FUNCTION_BLOCK FB_HVPS EXTENDS FB_HMIBase
VAR
	hvps : REFERENCE TO FB_HVPS_System;  // Reference to avoid copying and allow validation
	hvpsStatus : ARRAY[GC_HVPS.INDEX_SUPPLY_MIN..GC_HVPS.INDEX_SUPPLY_MAX] OF ST_HMIHvpsStatus;  // Status for all 4 supplies
END_VAR

METHOD ClearErrors : BOOL
VAR_INPUT
	index : DINT;
END_VAR
// Clear errors for specified supply
IF __ISVALIDREF(hvps) THEN
	hvps.ClearErrors(index);
	ClearErrors := TRUE;
END_IF
END_METHOD

METHOD Cyclic
VAR
	i : DINT;
	status : ARRAY[GC_HVPS.INDEX_SUPPLY_MIN..GC_HVPS.INDEX_SUPPLY_MAX] OF ST_PowerSupplyStatus;
END_VAR
// Sync status for each supply

// Check if HVPS reference is valid before accessing
IF NOT __ISVALIDREF(hvps) THEN
	RETURN;
END_IF

status := hvps.P_supplies_status;

FOR i := GC_HVPS.INDEX_SUPPLY_MIN TO GC_HVPS.INDEX_SUPPLY_MAX DO
	// Map HVPS-specific scalar status fields
	hvpsStatus[i].HmiStatus.Enabled := status[i].ENABLED;
	hvpsStatus[i].V_cur := status[i].VMON;
	hvpsStatus[i].I_cur := status[i].IMON;
	hvpsStatus[i].V_set := status[i].VSET;
	hvpsStatus[i].I_set := status[i].ISET;

	// Map base component status if reference is valid
	IF __ISVALIDREF(status[i].BaseComponentStatus) THEN
		hvpsStatus[i].HmiStatus.Busy := status[i].BaseComponentStatus.BaseStatus.Busy;
		hvpsStatus[i].HmiStatus.Done := status[i].BaseComponentStatus.BaseStatus.Done;
		hvpsStatus[i].HmiStatus.Error := status[i].BaseComponentStatus.BaseStatus.Error;
		hvpsStatus[i].HmiStatus.ErrorID := UDINT_TO_BYTE(status[i].BaseComponentStatus.BaseStatus.ErrorID);
	END_IF

	// Set error flag for HVPS-specific error conditions
	IF status[i].OverVoltageSetpointError OR
	   status[i].OverMaxVoltageError OR
	   status[i].OverCurrentSetpointError OR
	   status[i].OverMaxCurrentError THEN
		hvpsStatus[i].HmiStatus.Error := TRUE;
	END_IF
END_FOR

// Handle commands from base class
IF cmd.Enable THEN
	EnableHV(0);
	cmd.Enable := FALSE;
END_IF

IF cmd.Disable THEN
	DisableHV(0);
	cmd.Disable := FALSE;
END_IF
END_METHOD

METHOD DisableHV : BOOL
VAR_INPUT
	index : DINT;
END_VAR
// Disable HV output for specified supply
IF __ISVALIDREF(hvps) THEN
	hvps.Disable_HV(index);
	DisableHV := TRUE;
END_IF
END_METHOD

METHOD EnableHV : BOOL
VAR_INPUT
	index : DINT;
END_VAR
// Enable HV output for specified supply
IF __ISVALIDREF(hvps) THEN
	hvps.Enable_HV(index);
	EnableHV := TRUE;
END_IF
END_METHOD

METHOD FullShutdown : BOOL
VAR
END_VAR
// Emergency shutdown of all supplies
IF __ISVALIDREF(hvps) THEN
	hvps.FullShutDown();
	FullShutdown := TRUE;
END_IF
END_METHOD

METHOD GetSupplyStatus : ST_HMIHvpsStatus
VAR_INPUT
	index : DINT;
END_VAR
// Return status for specified supply
IF index >= 0 AND index <= 3 THEN
	GetSupplyStatus := hvpsStatus[index];
END_IF
END_METHOD

METHOD FB_init : BOOL
VAR_INPUT
	bInitRetains : BOOL; // if TRUE, the retain variables are initialized (warm start / cold start)
	bInCopyCode : BOOL;  // if TRUE, the instance afterwards gets moved into the copy code (online change)
END_VAR
// Standard FB constructor - no custom initialization needed
END_METHOD

METHOD Init : BOOL
VAR_INPUT
	refHVPS : REFERENCE TO FB_HVPS_System;
END_VAR
hvps REF= refHVPS;
Init := TRUE;
END_METHOD

// Property to access status of all 4 supplies
PROPERTY P_AllSupplyStatus : REFERENCE TO ARRAY[GC_HVPS.INDEX_SUPPLY_MIN..GC_HVPS.INDEX_SUPPLY_MAX] OF ST_HMIHvpsStatus
GET
P_AllSupplyStatus REF= hvpsStatus;
END_GET
END_PROPERTY

METHOD PowerOff : BOOL
VAR_INPUT
	index : DINT;
END_VAR
// Turn off input power to specified supply
IF __ISVALIDREF(hvps) THEN
	hvps.InputPowerOff(index);
	PowerOff := TRUE;
END_IF
END_METHOD

METHOD PowerOn : BOOL
VAR_INPUT
	index : DINT;
END_VAR
// Turn on input power to specified supply
IF __ISVALIDREF(hvps) THEN
	hvps.InputPowerOn(index);
	PowerOn := TRUE;
END_IF
END_METHOD

METHOD SetCurrent : BOOL
VAR_INPUT
	setpoint : LREAL;  // mA
	index : DINT;
END_VAR
// Set current setpoint for specified supply
IF __ISVALIDREF(hvps) THEN
	hvps.SetCurrent(setpoint, index);
	SetCurrent := TRUE;
END_IF
END_METHOD

METHOD SetVoltage : BOOL
VAR_INPUT
	setpoint : LREAL;  // V
	index : DINT;
END_VAR
// Set voltage setpoint for specified supply
IF __ISVALIDREF(hvps) THEN
	hvps.SetVoltage(setpoint, index);
	SetVoltage := TRUE;
END_IF
END_METHOD

END_FUNCTION_BLOCK

(* stored: Version 1.1.0.1
   POU FB_HVPS: Id {67ddd066-03fd-42be-8807-cd57f0c77bda}, SpecialFunc None
   Method ClearErrors: Id {f7a2b3c4-d5e6-47f8-9a0b-1c2d3e4f5a6b}
   Method Cyclic: Id {71ec0170-2f44-46d1-ad14-592c83aae3f9}
   Method DisableHV: Id {1098e173-96c7-4796-a7f2-193ef63a02a9}
   Method EnableHV: Id {325e924a-2d47-4a43-b44c-a3a640a61791}
   Method FullShutdown: Id {a1b2c3d4-e5f6-4789-0abc-def123456789}
   Method GetSupplyStatus: Id {e814ad49-555a-4e3e-afa8-48c2e8afba49}
   Method FB_init: Id {a53bc3e6-3670-4569-bfd0-dbbd953f4edc}
   Method Init: Id {a53bc3e7-3670-4569-bfd0-dbbd953f4edc}
   Property P_AllSupplyStatus: Id {b2c3d4e5-f6a7-4890-bcde-f012345678ab}
   Get Get: Id {c3d4e5f6-a789-4901-cdef-0123456789bc}
   Method PowerOff: Id {6f82d71a-8278-47c0-b837-4668c1bdeb51}
   Method PowerOn: Id {b234f18f-74f1-481d-91df-a10bda785615}
   Method SetCurrent: Id {f6ad2c9c-021f-470f-93d0-10c1bf54c683}
   Method SetVoltage: Id {eeff0e70-6255-427e-8a66-154b19c8c1bc} *)
